# EPICS StreamDevice protocol: air.proto
# Daedalus Air Quality Sensor protocol sensor file
# Built by modeling the Sidekick EPICS files

Terminator = CR LF;

# this method is used to retrieve the information for a specific sensor module
info {
	ExtraInput = Ignore;
	out "ID?";
	in "%39c";
}

# retrieving co2 data
getCO2 {
	out "Co2";
	in "%u";
}

# retrieving temperature data
getTemp {
	out "Temp";
	in "%f";
}

#retrieving humidity data
getHumi {
	out "Humi";
	in "%f";
}

debug {
   ExtraInput = Ignore;
   out "%s";
   in "%39c";
}
